PROGRAM G7_Palpage_Capacitance	
VAR_INPUT	SFCInit:BOOL;	END_VAR
VAR	SFCCurrentStep : STRING;	 	
	Ton_Step_11: TON;
	memo_besoin_decalage : BOOL := FALSE;
	RE_fct_palpage_seul	:R_TRIG;
	Re_Detect_Piece: R_trig;
	FE_Detect_Piece: F_trig;
	Memo_avant_decal_X : LREAL;
	Pas_besoin_palpage	:BOOL;
	floppytest	:BOOL;
END_VAR

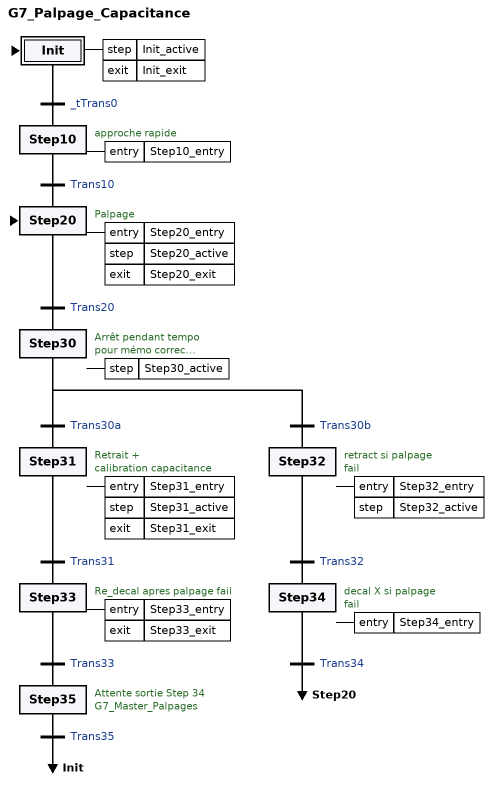
INITIAL_STEP Init:
    Init_active(N);  // step action
    Init_exit(P0);  // exit action
END_STEP
TRANSITION FROM Init TO Step10
    := _tTrans0;
END_TRANSITION
// approche rapide
STEP Step10:
    Step10_entry(P1);  // entry action
END_STEP
TRANSITION FROM Step10 TO Step20
    := Trans10;
END_TRANSITION
// Palpage
STEP Step20:
    Step20_entry(P1);  // entry action
    Step20_active(N);  // step action
    Step20_exit(P0);  // exit action
END_STEP
TRANSITION FROM Step20 TO Step30
    := Trans20;
END_TRANSITION
// Arrêt pendant tempo
// pour mémo correct
// +Test
STEP Step30:
    Step30_active(N);  // step action
END_STEP
TRANSITION FROM Step30 TO Step31
    := Trans30a;
END_TRANSITION
// Retrait +
// calibration capacitance
STEP Step31:
    Step31_entry(P1);  // entry action
    Step31_active(N);  // step action
    Step31_exit(P0);  // exit action
END_STEP
TRANSITION FROM Step31 TO Step33
    := Trans31;
END_TRANSITION
// Re_decal apres palpage fail
STEP Step33:
    Step33_entry(P1);  // entry action
    Step33_exit(P0);  // exit action
END_STEP
TRANSITION FROM Step30 TO Step32
    := Trans30b;
END_TRANSITION
// retract si palpage
// fail
STEP Step32:
    Step32_entry(P1);  // entry action
    Step32_active(N);  // step action
END_STEP
TRANSITION FROM Step32 TO Step34
    := Trans32;
END_TRANSITION
// decal X si palpage
// fail
STEP Step34:
    Step34_entry(P1);  // entry action
END_STEP
TRANSITION FROM Step34 TO Step20
    := Trans34;
END_TRANSITION
TRANSITION FROM Step33 TO Step35
    := Trans33;
END_TRANSITION
// Attente sortie Step 34
// G7_Master_Palpages
STEP Step35:
END_STEP
TRANSITION FROM Step35 TO Init
    := Trans35;
END_TRANSITION

TRANSITION _tTrans0:
 RE_Fct_palpage_Etal.Q OR (auto AND G7_Master_Palpages.step34.x)
END_TRANSITION

ACTION Init_active:
RE_fct_palpage_seul(clk:=Fct_palpage_Etal);
Prog_Start_Capacitance_Calibration:=false;
END_ACTION

ACTION Init_exit:
memo_besoin_decalage := FALSE;
Memo_X_Laser_Decal:=0;
END_ACTION

ACTION Step10_entry:
Pos_cible_Z_Laser:= Pnc_axe_Z_Robot.Limite_Plus-EP_Aile-30;	

IF Vitesse_approche_rapide > Pnc_axe_Z_Robot.Vitesse_PTP THEN
	Vitesse_Z_Laser_PTP:=Pnc_axe_Z_Robot.Vitesse_PTP;
ELSE
	Vitesse_Z_Laser_PTP:=Vitesse_approche_rapide;
END_IF
En_pos_Z_Laser:=false;
Top_Z_Laser:=TRUE;
END_ACTION

ACTION Step20_active:
Re_Detect_Piece(clk :=
	Data01_Capacitance_Actual_Value < 1); //UDINT valeur max 4 294 967 295, Buse en contact : detection capacitance (aug si dist baisse))
	
IF Re_Detect_Piece.Q THEN
	Pos_ref_torche_RE := Pos_Reel_Z_Laser - Axe_5.NcToPlc.PosDiff;
END_IF

(*//debug redondance top torche
IF NOT Top_Z_Laser AND No_Move_Z_Laser 
AND Data01_Capacitance_Actual_Value >2000000
AND Axe_5.NcToPlc.PosDiff<0.5 THEN
	Top_Z_Laser:=TRUE;
END_IF*)
END_ACTION

ACTION Step20_entry:
limite_couple_negatif_axe_Z_Laser :=LREAL_TO_INT(Couple_de_Palpage);

Pos_cible_Z_Laser:=Pnc_axe_Z_Robot.Limite_Plus-0.5;
IF Vitesse_de_palpage > Pnc_axe_Z_Robot.Vitesse_PTP THEN
	Vitesse_Z_Laser_PTP:=Pnc_axe_Z_Robot.Vitesse_PTP;
ELSE
	Vitesse_Z_Laser_PTP:=Vitesse_de_palpage;
END_IF
En_pos_Z_Laser:=FALSE;
Top_Z_Laser:=TRUE;
END_ACTION

ACTION Step20_exit:
Top_Z_Laser := FALSE;
limite_couple_negatif_axe_Z_Laser := 1000;
END_ACTION

ACTION Step30_active:
// Si palpage raté ...
IF NOT DI01_Collision AND Data01_Capacitance_Actual_Value > 2000000 THEN
	// ... alors on se décale pour ressayer.
	IF NOT memo_besoin_decalage  AND auto THEN
		Memo_avant_decal_X := Pos_Reel_X_Laser;
		memo_besoin_decalage := TRUE;
	// ... si décalage déjà testé, ...
	ELSE
		// ... alors on passe en défaut
		Test_capacitance_defectueux := TRUE;
		memo_besoin_decalage := FALSE;
	END_IF
END_IF
END_ACTION

ACTION Step31_active:
FE_Detect_Piece(clk :=Data01_Capacitance_Actual_Value < 2000000)	;
	
IF FE_Detect_Piece.Q THEN
	Pos_ref_torche_Fe := Pos_Reel_Z_Laser;
	Prog_Start_Capacitance_Calibration:=TRUE;	//Lors du retrait de la buse, on enregistre la capacitance dans un tableau selon la distance buse
END_IF

Prog_Distance_Buse_Piece_mm:= Pos_ref_torche_Fe - Pos_Reel_Z_Laser;
END_ACTION

ACTION Step31_entry:
Pos_ref_torche := Pos_ref_torche_RE;
//Pv_Z_Laser := TRUE;

Pos_cible_Z_Laser:=Pos_Reel_Z_Laser - 55;
IF Vitesse_de_palpage > Pnc_axe_Z_Robot.Vitesse_PTP THEN
	Vitesse_Z_Laser_PTP:=Pnc_axe_Z_Robot.Vitesse_PTP;
ELSE
	Vitesse_Z_Laser_PTP:=Vitesse_de_palpage/3;
END_IF
En_pos_Z_Laser:=FALSE;
Top_Z_Laser:=TRUE;
END_ACTION

ACTION Step31_exit:
Top_Z_Laser:=FALSE;

Pos_ref_torche := Pos_ref_torche_FE;

Palpage_Torche := FALSE;
Pv_Z_Laser := false;
END_ACTION

ACTION Step32_active:
IF NOT Top_Z_Laser AND NOT En_pos_Z_Laser THEN
	Top_Z_Laser:=TRUE;
END_IF
END_ACTION

ACTION Step32_entry:
Pos_cible_Z_Laser:=Pnc_axe_Z_Robot.Limite_moins+10;
Vitesse_Z_Laser_PTP:= Pnc_axe_Z_Robot.Vitesse_PTP;
Top_Z_Laser:=TRUE;
END_ACTION

ACTION Step33_entry:
IF memo_besoin_decalage THEN
 Pos_cible_X_Laser:=Memo_X_Laser_Decal;
 Top_X_Laser:=TRUE;
END_IF
END_ACTION

ACTION Step33_exit:
Nv_ProcessID := false;
END_ACTION

ACTION Step34_entry:
IF auto THEN //A affiner, revoir quels décals faire ? que X, ou aussi Y ? 
	// si auto, on decale en X
	Memo_X_Laser_Decal:=Pos_Reel_X_Laser;
	Pos_cible_X_Laser:=Pos_Reel_X_Laser +5;		
	Top_X_Laser:=TRUE;		
END_IF
END_ACTION

TRANSITION Trans10:
(
 (En_pos_Z_Laser AND NOT Top_Z_Laser AND No_Move_Z_Laser)
 //OR
 //(Pos_cible_Z_Laser>=Pnc_axe_Z_Robot.Limite_Plus-EP_Aile-ep_secu)
)
AND Step10.t>T#1S
END_TRANSITION

TRANSITION Trans20:
Data01_Capacitance_Actual_Value < 1
OR Axe_5.NcToPlc.PosDiff>=0.5
END_TRANSITION

TRANSITION Trans30a:
Step30.t > T#50MS	
AND No_Move_Z_Laser	
AND not memo_besoin_decalage
END_TRANSITION

TRANSITION Trans30b:
Step30.t > T#50MS	
AND No_Move_Z_Laser	
AND memo_besoin_decalage
END_TRANSITION

TRANSITION Trans31:
Data01_Capacitance_Actual_Value > 2000000
AND Prog_Capacitance_Calibration_OK
AND NOT Top_Z_Laser
AND En_pos_Z_Laser
AND No_Move_Z_Laser
AND step31.t > T#20MS
END_TRANSITION

TRANSITION Trans32:
Step32.t > T#50MS
AND En_pos_Z_Laser 
AND NOT Top_Z_Laser 
AND No_Move_Z_Laser
END_TRANSITION

TRANSITION Trans33:
NOT Fct_palpage_Etal
AND

	En_pos_Z_Laser AND NOT Top_Z_Laser
	AND No_Move_Z_Laser
	AND En_pos_X_Laser AND NOT Top_X_Laser
	AND No_Move_X_Laser
END_TRANSITION

TRANSITION Trans34:
memo_besoin_decalage
AND	auto 
AND Step34.t>T#20MS
AND(NOT Top_X_Laser AND En_pos_X_Laser )
END_TRANSITION

TRANSITION Trans35:
not G7_Master_Palpages.step34.x
END_TRANSITION

END_PROGRAM

(* stored: Version 1.1.0.1
   POU G7_Palpage_Capacitance: Id {8bf53146-8e83-4680-baef-2f82619e572c}, SpecialFunc None
   Transition _tTrans0: Id {fda42855-65ce-49b2-aebd-a27fb3b765b8}
   Action Init_active: Id {6c6b803e-94fe-4973-a3db-39b3b6ea881f}
   Action Init_exit: Id {e3d2b9e0-19e0-446f-9109-9f68deddd8da}
   Action Step10_entry: Id {ec80f881-c879-4eb0-b9db-b55a4c9ffcdd}
   Action Step20_active: Id {f926592e-8b95-49c1-9273-718b7a84803d}
   Action Step20_entry: Id {53bbef7f-5647-4459-9bdf-9cba9d586bed}
   Action Step20_exit: Id {877be295-a8ac-435f-96ce-d7bfaf4a9380}
   Action Step30_active: Id {a4aab25e-dc53-4305-9940-e0a275e3fa42}
   Action Step31_active: Id {9642a9b0-90c3-44ac-b540-31fffc53a98d}
   Action Step31_entry: Id {cca5c4e9-2974-426b-9f8c-b20bf5e377a2}
   Action Step31_exit: Id {23e98cc3-a4a6-46a0-9c0a-21b2c089844c}
   Action Step32_active: Id {b4bc66b8-0043-4d67-ab55-1d3b5715f46c}
   Action Step32_entry: Id {232abdcb-02b9-4431-92df-28882fac747c}
   Action Step33_entry: Id {63611fc7-1840-4078-85f8-960782d246d4}
   Action Step33_exit: Id {90643c6a-70d8-4c31-9110-a6c29389a67a}
   Action Step34_entry: Id {5c0f5f85-6f8c-4e71-a40d-b3dda79df7cf}
   Transition Trans10: Id {4d78375c-a38d-41bb-9a13-b56b5311ab70}
   Transition Trans20: Id {b3433e34-56a0-482d-a145-cf017a5dc98e}
   Transition Trans30a: Id {aa446346-44ec-4010-a73a-9349e7783501}
   Transition Trans30b: Id {93f30dee-1157-48e3-88b5-c83c0e7cda8b}
   Transition Trans31: Id {37d2d310-4e23-482a-a051-513dbd809572}
   Transition Trans32: Id {dc47ac83-ec16-4ed1-96ad-4a2efc21c4a0}
   Transition Trans33: Id {2032d5a5-78c5-404c-8d30-e4aef03160ce}
   Transition Trans34: Id {6b014c8d-ff73-4cdd-a278-f5b0968f6c8c}
   Transition Trans35: Id {c12af936-c4a5-468c-b35f-a6da67fcfdaa} *)
